FUNCTION_BLOCK PUBLIC FB_ALARM
VAR_IN_OUT
	Handler : FB_ALARM_HANDLER;
END_VAR
VAR_INPUT
	Config : TYP_ALARM_CONFIG;
END_VAR
VAR_OUTPUT
	State : E_ALARM_STATE;
END_VAR

METHOD PUBLIC Acknowledge : REFERENCE TO FB_ALARM
VAR_INPUT
END_VAR
VAR
	PreviousState : E_ALARM_STATE;
END_VAR
{warning disable C0371}

// Checking the VAR_IN_OUT reference, leave the current method in case of invalid reference
IF NOT __ISVALIDREF(THIS^.Handler) THEN
     RETURN;
END_IF


PreviousState := THIS^.State;

CASE THIS^.State OF 
	
	E_ALARM_STATE.ACTIVE_UNACK:
	
		CASE THIS^.Config.Acknowledge OF
			
			E_ALARM_ACK_TYPE.ONLY_ACK:
				THIS^.State := E_ALARM_STATE.INACTIVE;
				
			E_ALARM_ACK_TYPE.ACK_OR_RESET:
				THIS^.State := E_ALARM_STATE.INACTIVE;
			
			E_ALARM_ACK_TYPE.ACK_AFTER_RESET:
				;
				
			ELSE
				THIS^.State := E_ALARM_STATE.ACTIVE_ACK;
			
		END_CASE;

	E_ALARM_STATE.INACTIVE_UNACK:
		
		THIS^.State := E_ALARM_STATE.INACTIVE;
					
	ELSE
		;
		
END_CASE;

IF THIS^.State <> PreviousState THEN
	THIS^.Handler.RegisterAlarm(Alarm := THIS^, Prefix := '', Update := TRUE);
END_IF;

Acknowledge REF= THIS^;
END_METHOD

METHOD PUBLIC AcknowledgeNoUpdate : REFERENCE TO FB_ALARM
VAR_INPUT
END_VAR
VAR
	PreviousState : E_ALARM_STATE;
END_VAR
{warning disable C0371}

// Checking the VAR_IN_OUT reference, leave the current method in case of invalid reference
IF NOT __ISVALIDREF(THIS^.Handler) THEN
     RETURN;
END_IF


PreviousState := THIS^.State;

CASE THIS^.State OF 
	
	E_ALARM_STATE.ACTIVE_UNACK:
	
		CASE THIS^.Config.Acknowledge OF
			
			E_ALARM_ACK_TYPE.ONLY_ACK:
				THIS^.State := E_ALARM_STATE.INACTIVE;
				
			E_ALARM_ACK_TYPE.ACK_OR_RESET:
				THIS^.State := E_ALARM_STATE.INACTIVE;
			
			E_ALARM_ACK_TYPE.ACK_AFTER_RESET:
				;
				
			ELSE
				THIS^.State := E_ALARM_STATE.ACTIVE_ACK;
			
		END_CASE;

	E_ALARM_STATE.INACTIVE_UNACK:
		
		THIS^.State := E_ALARM_STATE.INACTIVE;
					
	ELSE
		;
		
END_CASE;

IF THIS^.State <> PreviousState THEN
	THIS^.Handler.RegisterAlarm(Alarm := THIS^, Prefix := '', Update := FALSE);
END_IF;

AcknowledgeNoUpdate REF= THIS^;
END_METHOD

METHOD PUBLIC Activate : REFERENCE TO FB_ALARM
VAR_INPUT
END_VAR
VAR
	PreviousState : E_ALARM_STATE;
END_VAR
{warning disable C0371}

// Checking the VAR_IN_OUT reference, leave the current method in case of invalid reference
IF NOT __ISVALIDREF(THIS^.Handler) THEN
     RETURN;
END_IF


PreviousState := THIS^.State;

CASE THIS^.State OF 
	
	E_ALARM_STATE.ACTIVE_ACK:
		// Keeps the state as active and acknowledged
		;
			
	ELSE
		// Any other state will turn it into active and unacknowledged
		THIS^.State := E_ALARM_STATE.ACTIVE_UNACK;
		
END_CASE;

IF THIS^.State <> PreviousState THEN
	THIS^.Handler.RegisterAlarm(Alarm := THIS^, Prefix := '', Update := TRUE);
END_IF;

Activate REF= THIS^;
END_METHOD

PROPERTY PUBLIC IsActive : BOOL
GET
IsActive := THIS^.State = E_ALARM_STATE.ACTIVE_ACK OR THIS^.State = E_ALARM_STATE.ACTIVE_UNACK;
END_GET
END_PROPERTY

METHOD PUBLIC Reset : REFERENCE TO FB_ALARM
VAR_INPUT
END_VAR
VAR
	PreviousState : E_ALARM_STATE;
END_VAR
{warning disable C0371}

// Checking the VAR_IN_OUT reference, leave the current method in case of invalid reference
IF NOT __ISVALIDREF(THIS^.Handler) THEN
     RETURN;
END_IF


PreviousState := THIS^.State;

CASE THIS^.State OF 
	
	E_ALARM_STATE.ACTIVE_UNACK:
	
		CASE THIS^.Config.Acknowledge OF
			
			E_ALARM_ACK_TYPE.ONLY_RESET:
				THIS^.State := E_ALARM_STATE.INACTIVE;
				
			E_ALARM_ACK_TYPE.ACK_OR_RESET:
				THIS^.State := E_ALARM_STATE.INACTIVE;
				
			ELSE
				THIS^.State := E_ALARM_STATE.INACTIVE_UNACK;
			
		END_CASE;
		
	E_ALARM_STATE.ACTIVE_ACK:
		THIS^.State := E_ALARM_STATE.INACTIVE;
			
	ELSE
		;
		
END_CASE;

IF THIS^.State <> PreviousState THEN
	THIS^.Handler.RegisterAlarm(Alarm := THIS^, Prefix := '', Update := TRUE);
END_IF;

Reset REF= THIS^;
END_METHOD

END_FUNCTION_BLOCK

(* stored: Version 1.1.0.1, ProductVersion 3.1.4024.12
   POU FB_ALARM: Id {a9f298f4-ca32-450c-a79c-fc4266c53d1d}, SpecialFunc None
   Method Acknowledge: Id {00199362-b98d-451a-be12-3d64270740b1}
   Method AcknowledgeNoUpdate: Id {07562f46-cb18-4f39-ad81-bdeccc127250}
   Method Activate: Id {165d8d33-ea10-4d15-87ae-5005372ac614}
   Property IsActive: Id {8925a5ee-41cc-4f64-adb7-4a3115971f9f}
   Get Get: Id {523c8c41-fc0b-4eb3-b34b-556dce47cb2a}
   Method Reset: Id {7bb42957-5629-472c-9636-6a4199d056cc} *)
